(* Logix 5000 project; controller Amvex_Thorpe_Flowmeter vendor 1 type 14 code 106 rev 33.13; software revision 33.01; part 10 of 16 *)
(* tags used below, declared in another part *)
   FIRST_SCAN : BOOL;
   FIRST_SCAN_ONS : BOOL;
   ID86_InputDataLength : MESSAGE;   // Message Command Input Data Data Length
   ID86_LengthParameterdata : MESSAGE;   // Message Command Parameter Data Length
   ID86_MSG_Diagnostic : MESSAGE;   // Message Get Diagnosis Module
   ID86_MSG_ProcessAlarm : MESSAGE;   // Message Get Get Process Alram Module
   ID86_OutputDataLength : MESSAGE;   // Message Command Output Data Data Length
   ID86_ReceiveMSG1 : MESSAGE;   // Message Command Parameter Receive Data
   ID86_ReceiveMSG2 : MESSAGE;   // Message Command Parameter Receive Data
   ID86_ReceiveMSG3 : MESSAGE;   // Message Command Parameter Receive Data
   ID86_SendMSG1 : MESSAGE;   // Message Command Parameter Send Data
   ID86_SendMSG2 : MESSAGE;   // Message Command Parameter Send Data
   ID86_SendMSG3 : MESSAGE;   // Message Command Parameter Send Data
   MCP_00 : UDT_ID86;

PROGRAM MainProgram   (* main routine MainRoutine *)
VAR
   test : INT := 8;
END_VAR

ROUTINE MainRoutine   (* ladder *)
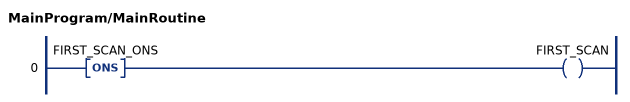
   0: ONS(FIRST_SCAN_ONS)OTE(FIRST_SCAN);
END_ROUTINE
END_PROGRAM

PROGRAM MCP_Main   (* main routine MAIN *)
VAR
   ActivateBtn : BOOL;
   Alicat0_ONS : BOOL;
   Alicat0DataInc : INT := 2;
   Alicat1_ONS : BOOL;
   Alicat1_ONS2 : BOOL := 1;
   Alicat1DataInc : INT := 7;
   Auto_Seq : SEQ := (Time_Out.PRE := 180000, Time_Out.ACC := 114179, Time_Out.EN := 1, Time_Out.TT := 1, Time_Out_Sec := 180);
   Barcode_Latch : BOOL;
   Barcode_ONS : BOOL;
   Barcode_Result_DATA : SINT[128] := ([0] := 69, [1] := 82, [2] := 82, [3] := 79, [4] := 82, [5] := 13, [6] := 56, [7] := 49, [8] := 48, [9] := 49, [10] := 53, [11] := 48, [12] := 51, [13] := 48, [14] := 48, [15] := 48, [16] := 50, [17] := 49, [18] := 84, [19] := 49, [20] := 53, [21] := 85, [22] := 79, [23] := 66, [24] := 51, [25] := 53, [26] := 48, [27] := 57, [28] := 56, [29] := 13);
   BarcodeSave_ons : BOOL;
   Counter_ONS : BOOL;
   debugtimer1 : TIMER := (PRE := 1000);
   DonePallets : COUNTER := (ACC := -70770);
   Fasttest_timer : TIMER := (PRE := 750);
   Fasttest_timer2 : TIMER := (PRE := 1000);
   FAULT : DINT;
   FAULTED : DINT;
   First_SEQ : BOOL;
   First_SEQ_ONS : BOOL;
   Flash_Timer_Off : TIMER := (PRE := 500);
   Flash_Timer_On : TIMER := (PRE := 500, ACC := 430, EN := 1, TT := 1);
   Gripper_ONS : BOOL;
   HMI_Counter_ONS : BOOL;
   Home_ONS : BOOL;
   HomeStep : INT;
   Infeed_Latch : BOOL;
   Infeed_ONS : BOOL := 1;
   InfeedPalletTM1 : TIMER := (PRE := 250);
   InfeedPalletTM2 : TIMER := (PRE := 250);
   IV3_Prog_AOI : IvSwichPrgoram := (TargetProgramNo := 3, SwitchProgramDone := 1);
   joggingONS : BOOL;
   Lift_stop_timer : TIMER := (PRE := 750);
   lift_stop_timer2 : TIMER := (PRE := 750);
   Manual_ONS : BOOL;
   Manual_Output_Reset : BOOL;
   MODE : MODE := (Manual := 1, Manual_ONS := 1, Selector := 2);
   Oxygen_TM : TIMER := (PRE := 500);
   PalletStop_ONS : BOOL;
   Part_count : DINT := 39;
   Prog_Switch_ons : BOOL;
   RCD_ONS : BOOL;
   RESET : BOOL;
   Rest_timer : TIMER := (PRE := 1000);
   RobotAngVel : SetCartAngVel := (Parameter_Value := 50.0);
   RobotConnected_ONS : BOOL;
   RobotConnection : BOOL;
   Setspeed : BOOL;
   SetupONS : BOOL;
   SR_Read_Complete_Clear : BOOL;
   SR_Read_Request : BOOL;
   SR_ReadSuccess : BOOL;
   Stopping_Latch : BOOL := 1;
   temp_Gripper_Delay : TIMER := (PRE := 250);
   Test : Connect;
   Test_Connection : Connect;
   Test_ONS : BOOL[32];
   Test_start_offline : StartOfflineProgram := (Parameter_Value := 1.0);
   test_Turn_ONS : BOOL;
   testing_ons : BOOL;
   testsstse : BOOL;
END_VAR

ROUTINE MAIN   (* ladder *)
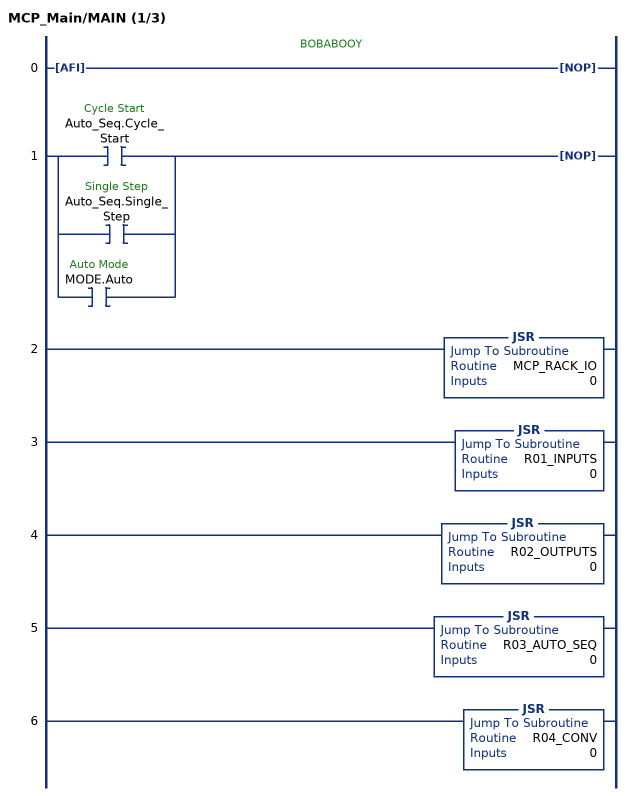
   // BOBABOOY
   0: AFI()NOP();
   1: [XIC(Auto_Seq.Cycle_Start) ,XIC(Auto_Seq.Single_Step) ,XIC(MODE.Auto) ]NOP();
   2: JSR(MCP_RACK_IO,0);
   3: JSR(R01_INPUTS,0);
   4: JSR(R02_OUTPUTS,0);
   5: JSR(R03_AUTO_SEQ,0);
   6: JSR(R04_CONV,0);
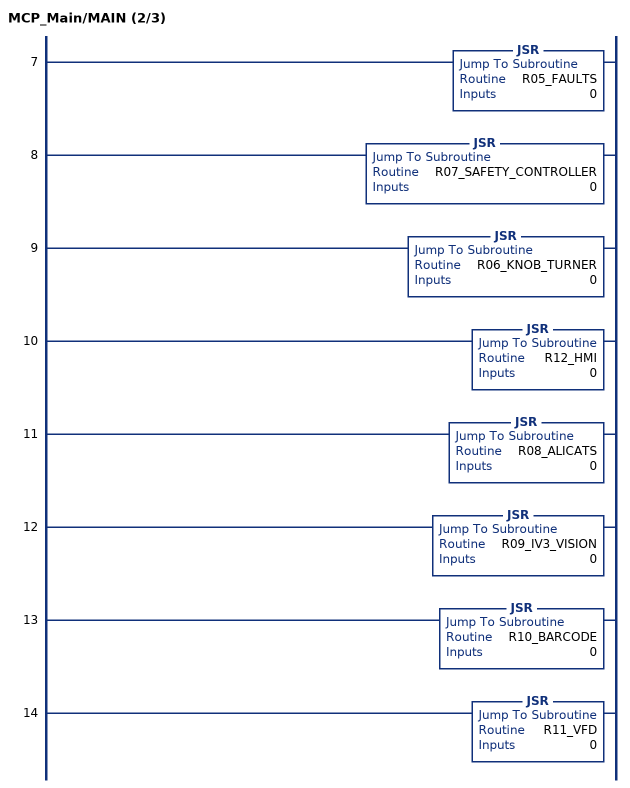
   7: JSR(R05_FAULTS,0);
   8: JSR(R07_SAFETY_CONTROLLER,0);
   9: JSR(R06_KNOB_TURNER,0);
   10: JSR(R12_HMI,0);
   11: JSR(R08_ALICATS,0);
   12: JSR(R09_IV3_VISION,0);
   13: JSR(R10_BARCODE,0);
   14: JSR(R11_VFD,0);
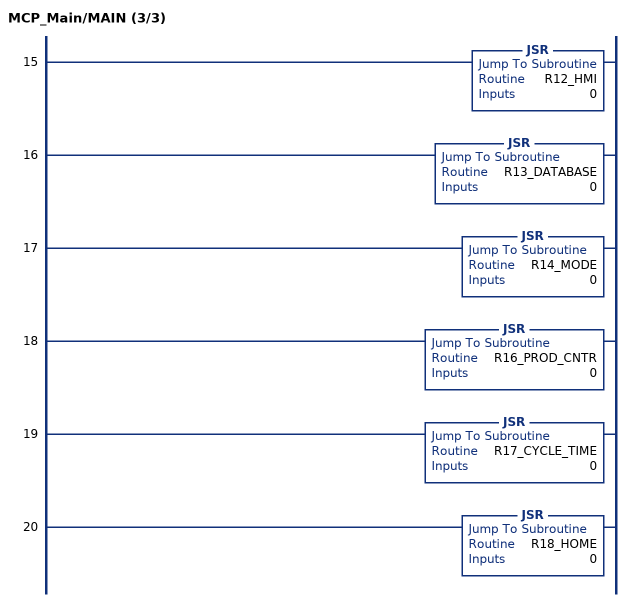
   15: JSR(R12_HMI,0);
   16: JSR(R13_DATABASE,0);
   17: JSR(R14_MODE,0);
   18: JSR(R16_PROD_CNTR,0);
   19: JSR(R17_CYCLE_TIME,0);
   20: JSR(R18_HOME,0);
END_ROUTINE

ROUTINE MCP_RACK_IO   (* ladder *)
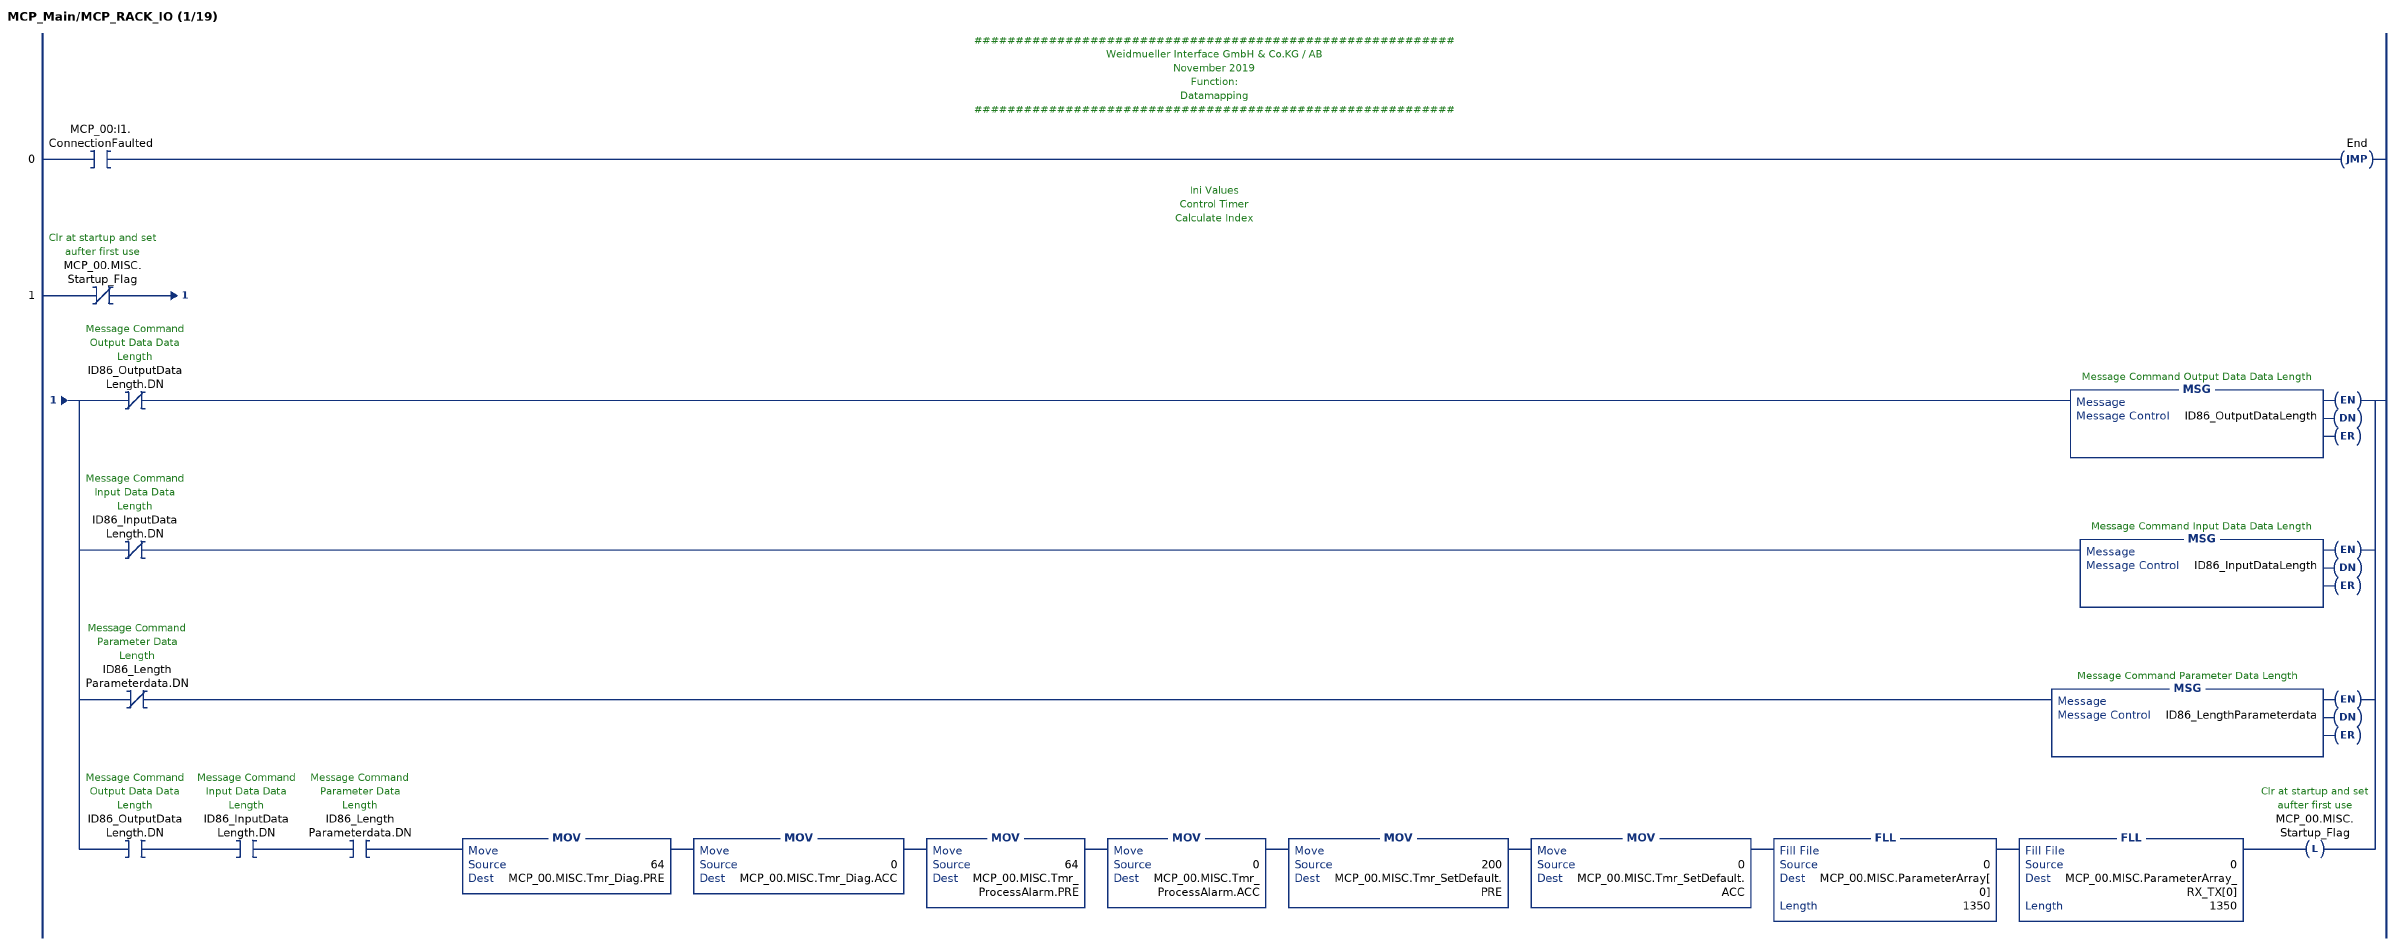
   // ##########################################################
   // Weidmueller Interface GmbH & Co.KG / AB
   // November 2019
   // Function:
   // Datamapping
   // ##########################################################
   0: XIC(MCP_00:I1.ConnectionFaulted)JMP(End);
   // Ini Values
   // Control Timer
   // Calculate Index
   1: XIO(MCP_00.MISC.Startup_Flag)[[XIO(ID86_OutputDataLength.DN) MSG(ID86_OutputDataLength) ,XIO(ID86_InputDataLength.DN) MSG(ID86_InputDataLength) ,XIO(ID86_LengthParameterdata.DN) MSG(ID86_LengthParameterdata) ] ,XIC(ID86_OutputDataLength.DN) XIC(ID86_InputDataLength.DN) XIC(ID86_LengthParameterdata.DN) MOV(64,MCP_00.MISC.Tmr_Diag.PRE) MOV(0,MCP_00.MISC.Tmr_Diag.ACC) MOV(64,MCP_00.MISC.Tmr_ProcessAlarm.PRE) MOV(0,MCP_00.MISC.Tmr_ProcessAlarm.ACC) MOV(200,MCP_00.MISC.Tmr_SetDefault.PRE) MOV(0,MCP_00.MISC.Tmr_SetDefault.ACC) FLL(0,MCP_00.MISC.ParameterArray[0],1350) FLL(0,MCP_00.MISC.ParameterArray_RX_TX[0],1350) OTL(MCP_00.MISC.Startup_Flag) ];
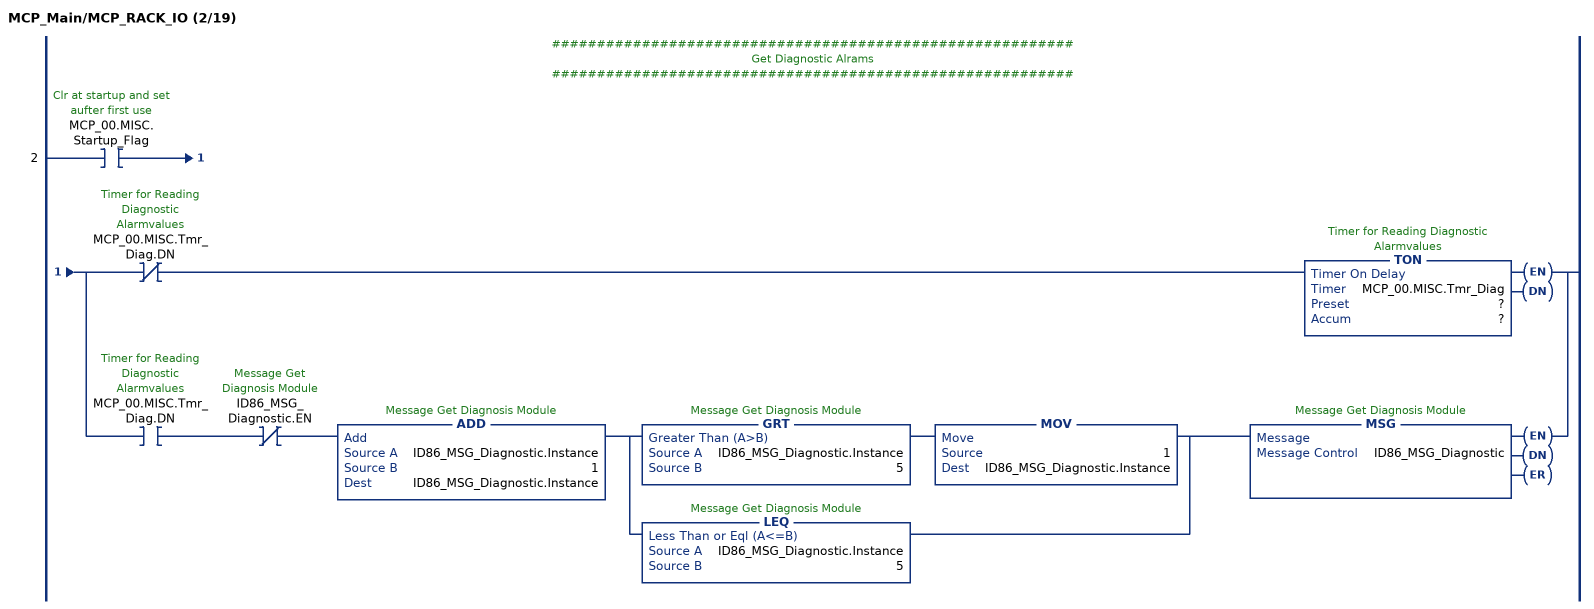
   // ##########################################################
   // Get Diagnostic Alrams
   // ##########################################################
   2: XIC(MCP_00.MISC.Startup_Flag)[XIO(MCP_00.MISC.Tmr_Diag.DN) TON(MCP_00.MISC.Tmr_Diag,?,?) ,XIC(MCP_00.MISC.Tmr_Diag.DN) XIO(ID86_MSG_Diagnostic.EN) ADD(ID86_MSG_Diagnostic.Instance,1,ID86_MSG_Diagnostic.Instance) [GRT(ID86_MSG_Diagnostic.Instance,5) MOV(1,ID86_MSG_Diagnostic.Instance) ,LEQ(ID86_MSG_Diagnostic.Instance,5) ] MSG(ID86_MSG_Diagnostic) ];
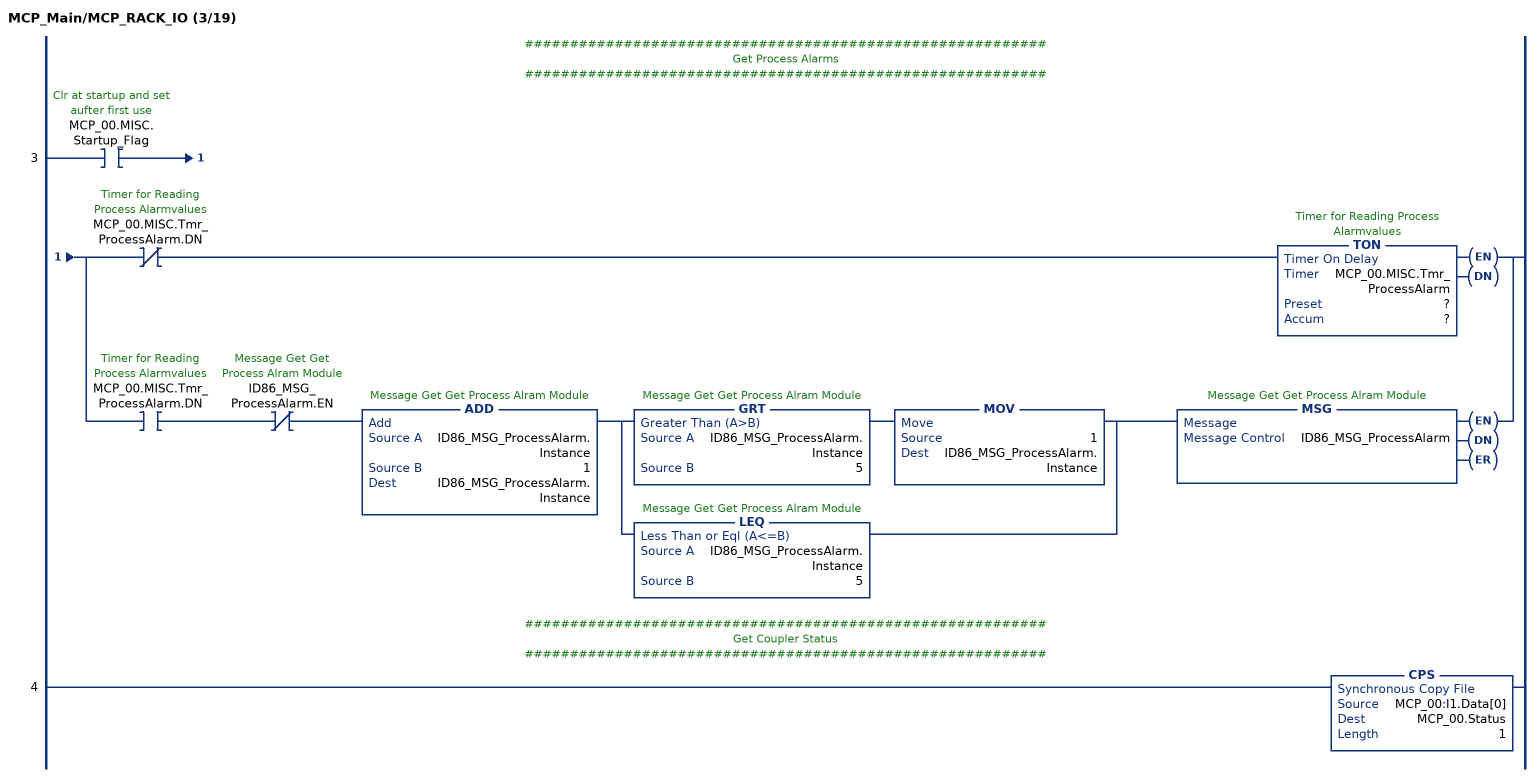
   // ##########################################################
   // Get Process Alarms
   // ##########################################################
   3: XIC(MCP_00.MISC.Startup_Flag)[XIO(MCP_00.MISC.Tmr_ProcessAlarm.DN) TON(MCP_00.MISC.Tmr_ProcessAlarm,?,?) ,XIC(MCP_00.MISC.Tmr_ProcessAlarm.DN) XIO(ID86_MSG_ProcessAlarm.EN) ADD(ID86_MSG_ProcessAlarm.Instance,1,ID86_MSG_ProcessAlarm.Instance) [GRT(ID86_MSG_ProcessAlarm.Instance,5) MOV(1,ID86_MSG_ProcessAlarm.Instance) ,LEQ(ID86_MSG_ProcessAlarm.Instance,5) ] MSG(ID86_MSG_ProcessAlarm) ];
   // ##########################################################
   // Get Coupler Status
   // ##########################################################
   4: CPS(MCP_00:I1.Data[0],MCP_00.Status,1);
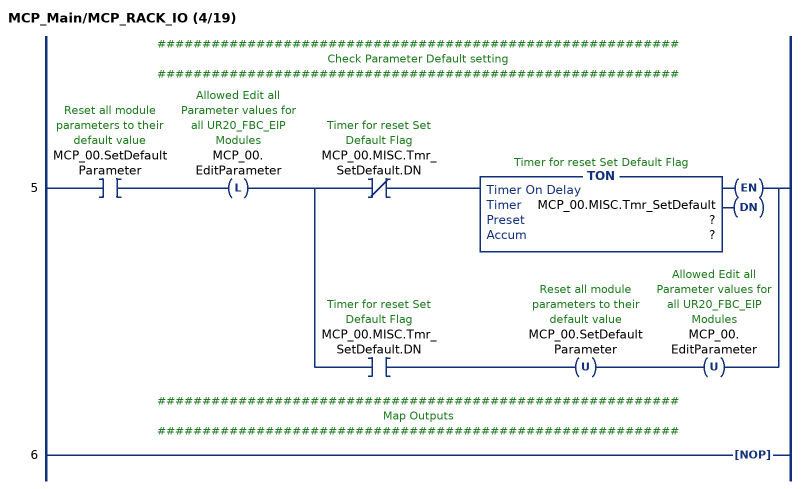
   // ##########################################################
   // Check Parameter Default setting
   // ##########################################################
   5: XIC(MCP_00.SetDefaultParameter)OTL(MCP_00.EditParameter)[XIO(MCP_00.MISC.Tmr_SetDefault.DN) TON(MCP_00.MISC.Tmr_SetDefault,?,?) ,XIC(MCP_00.MISC.Tmr_SetDefault.DN) OTU(MCP_00.SetDefaultParameter) OTU(MCP_00.EditParameter) ];
   // ##########################################################
   // Map Outputs
   // ##########################################################
   6: NOP();
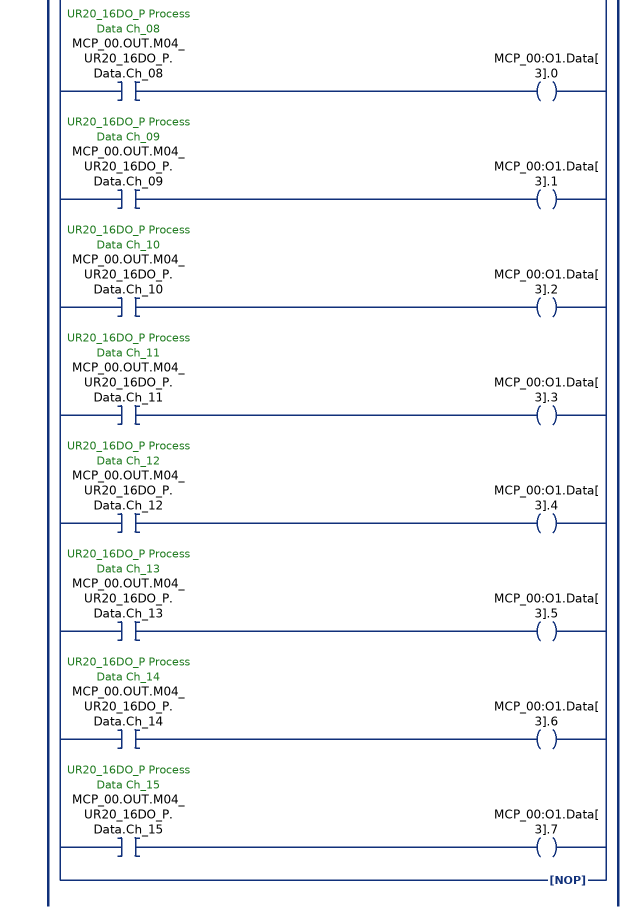
   // Map
   //  UR20_16DO_P
   //  Module No 4
   //  Process Data
   //  Outputs
   7: [NOP() ,XIC(MCP_00.OUT.M04_UR20_16DO_P.Data.Ch_00) OTE(MCP_00:O1.Data[2].0) ,XIC(MCP_00.OUT.M04_UR20_16DO_P.Data.Ch_01) OTE(MCP_00:O1.Data[2].1) ,XIC(MCP_00.OUT.M04_UR20_16DO_P.Data.Ch_02) OTE(MCP_00:O1.Data[2].2) ,XIC(MCP_00.OUT.M04_UR20_16DO_P.Data.Ch_03) OTE(MCP_00:O1.Data[2].3) ,XIC(MCP_00.OUT.M04_UR20_16DO_P.Data.Ch_04) OTE(MCP_00:O1.Data[2].4) ,XIC(MCP_00.OUT.M04_UR20_16DO_P.Data.Ch_05) OTE(MCP_00:O1.Data[2].5) ,XIC(MCP_00.OUT.M04_UR20_16DO_P.Data.Ch_06) OTE(MCP_00:O1.Data[2].6) ,XIC(MCP_00.OUT.M04_UR20_16DO_P.Data.Ch_07) OTE(MCP_00:O1.Data[2].7) ,XIC(MCP_00.OUT.M04_UR20_16DO_P.Data.Ch_08) OTE(MCP_00:O1.Data[3].0) ,XIC(MCP_00.OUT.M04_UR20_16DO_P.Data.Ch_09) OTE(MCP_00:O1.Data[3].1) ,XIC(MCP_00.OUT.M04_UR20_16DO_P.Data.Ch_10) OTE(MCP_00:O1.Data[3].2) ,XIC(MCP_00.OUT.M04_UR20_16DO_P.Data.Ch_11) OTE(MCP_00:O1.Data[3].3) ,XIC(MCP_00.OUT.M04_UR20_16DO_P.Data.Ch_12) OTE(MCP_00:O1.Data[3].4) ,XIC(MCP_00.OUT.M04_UR20_16DO_P.Data.Ch_13) OTE(MCP_00:O1.Data[3].5) ,XIC(MCP_00.OUT.M04_UR20_16DO_P.Data.Ch_14) OTE(MCP_00:O1.Data[3].6) ,XIC(MCP_00.OUT.M04_UR20_16DO_P.Data.Ch_15) OTE(MCP_00:O1.Data[3].7) ,NOP() ];
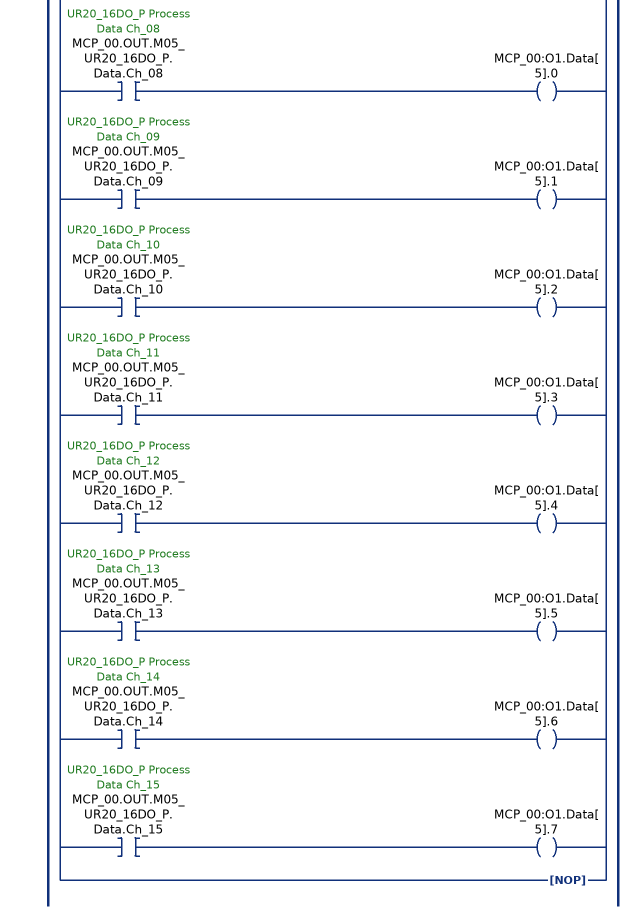
   // Map
   //  UR20_16DO_P
   //  Module No 5
   //  Process Data
   //  Outputs
   8: [NOP() ,XIC(MCP_00.OUT.M05_UR20_16DO_P.Data.Ch_00) OTE(MCP_00:O1.Data[4].0) ,XIC(MCP_00.OUT.M05_UR20_16DO_P.Data.Ch_01) OTE(MCP_00:O1.Data[4].1) ,XIC(MCP_00.OUT.M05_UR20_16DO_P.Data.Ch_02) OTE(MCP_00:O1.Data[4].2) ,XIC(MCP_00.OUT.M05_UR20_16DO_P.Data.Ch_03) OTE(MCP_00:O1.Data[4].3) ,XIC(MCP_00.OUT.M05_UR20_16DO_P.Data.Ch_04) OTE(MCP_00:O1.Data[4].4) ,XIC(MCP_00.OUT.M05_UR20_16DO_P.Data.Ch_05) OTE(MCP_00:O1.Data[4].5) ,XIC(MCP_00.OUT.M05_UR20_16DO_P.Data.Ch_06) OTE(MCP_00:O1.Data[4].6) ,XIC(MCP_00.OUT.M05_UR20_16DO_P.Data.Ch_07) OTE(MCP_00:O1.Data[4].7) ,XIC(MCP_00.OUT.M05_UR20_16DO_P.Data.Ch_08) OTE(MCP_00:O1.Data[5].0) ,XIC(MCP_00.OUT.M05_UR20_16DO_P.Data.Ch_09) OTE(MCP_00:O1.Data[5].1) ,XIC(MCP_00.OUT.M05_UR20_16DO_P.Data.Ch_10) OTE(MCP_00:O1.Data[5].2) ,XIC(MCP_00.OUT.M05_UR20_16DO_P.Data.Ch_11) OTE(MCP_00:O1.Data[5].3) ,XIC(MCP_00.OUT.M05_UR20_16DO_P.Data.Ch_12) OTE(MCP_00:O1.Data[5].4) ,XIC(MCP_00.OUT.M05_UR20_16DO_P.Data.Ch_13) OTE(MCP_00:O1.Data[5].5) ,XIC(MCP_00.OUT.M05_UR20_16DO_P.Data.Ch_14) OTE(MCP_00:O1.Data[5].6) ,XIC(MCP_00.OUT.M05_UR20_16DO_P.Data.Ch_15) OTE(MCP_00:O1.Data[5].7) ,NOP() ];
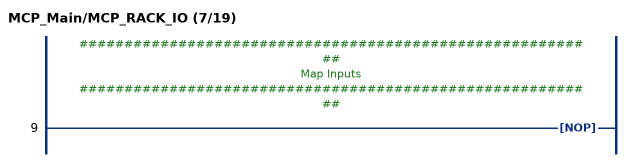
   // ##########################################################
   // Map Inputs
   // ##########################################################
   9: NOP();
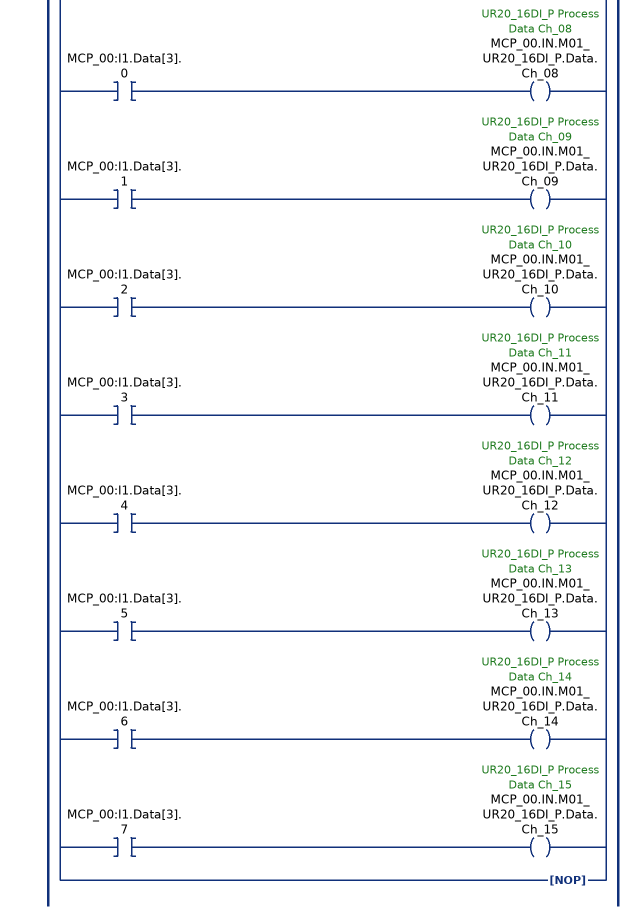
   // Map
   //  UR20_16DI_P
   //  Module No 1
   //  Process Data
   //  Inputs
   10: [NOP() ,XIC(MCP_00:I1.Data[2].0) OTE(MCP_00.IN.M01_UR20_16DI_P.Data.Ch_00) ,XIC(MCP_00:I1.Data[2].1) OTE(MCP_00.IN.M01_UR20_16DI_P.Data.Ch_01) ,XIC(MCP_00:I1.Data[2].2) OTE(MCP_00.IN.M01_UR20_16DI_P.Data.Ch_02) ,XIC(MCP_00:I1.Data[2].3) OTE(MCP_00.IN.M01_UR20_16DI_P.Data.Ch_03) ,XIC(MCP_00:I1.Data[2].4) OTE(MCP_00.IN.M01_UR20_16DI_P.Data.Ch_04) ,XIC(MCP_00:I1.Data[2].5) OTE(MCP_00.IN.M01_UR20_16DI_P.Data.Ch_05) ,XIC(MCP_00:I1.Data[2].6) OTE(MCP_00.IN.M01_UR20_16DI_P.Data.Ch_06) ,XIC(MCP_00:I1.Data[2].7) OTE(MCP_00.IN.M01_UR20_16DI_P.Data.Ch_07) ,XIC(MCP_00:I1.Data[3].0) OTE(MCP_00.IN.M01_UR20_16DI_P.Data.Ch_08) ,XIC(MCP_00:I1.Data[3].1) OTE(MCP_00.IN.M01_UR20_16DI_P.Data.Ch_09) ,XIC(MCP_00:I1.Data[3].2) OTE(MCP_00.IN.M01_UR20_16DI_P.Data.Ch_10) ,XIC(MCP_00:I1.Data[3].3) OTE(MCP_00.IN.M01_UR20_16DI_P.Data.Ch_11) ,XIC(MCP_00:I1.Data[3].4) OTE(MCP_00.IN.M01_UR20_16DI_P.Data.Ch_12) ,XIC(MCP_00:I1.Data[3].5) OTE(MCP_00.IN.M01_UR20_16DI_P.Data.Ch_13) ,XIC(MCP_00:I1.Data[3].6) OTE(MCP_00.IN.M01_UR20_16DI_P.Data.Ch_14) ,XIC(MCP_00:I1.Data[3].7) OTE(MCP_00.IN.M01_UR20_16DI_P.Data.Ch_15) ,NOP() ];
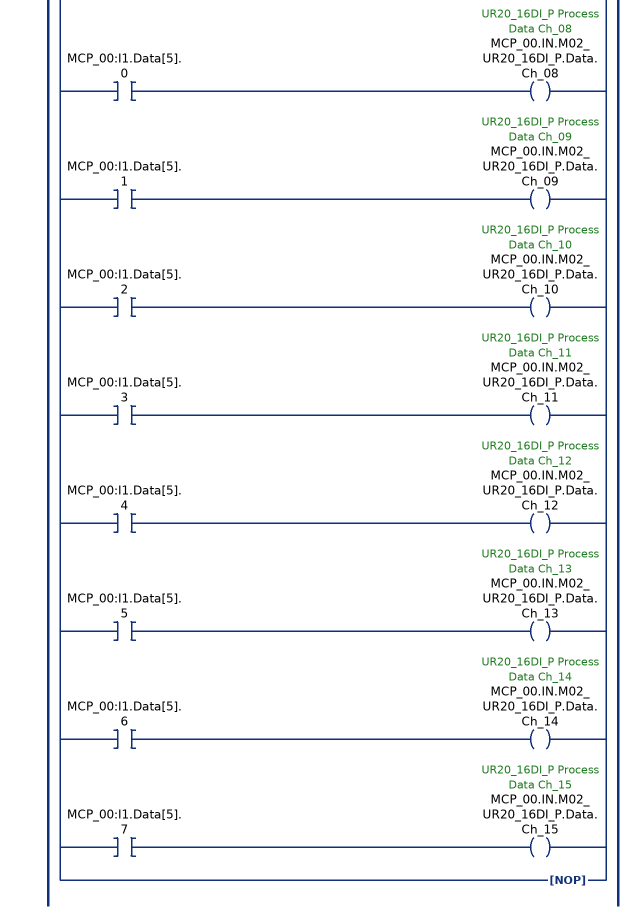
   // Map
   //  UR20_16DI_P
   //  Module No 2
   //  Process Data
   //  Inputs
   11: [NOP() ,XIC(MCP_00:I1.Data[4].0) OTE(MCP_00.IN.M02_UR20_16DI_P.Data.Ch_00) ,XIC(MCP_00:I1.Data[4].1) OTE(MCP_00.IN.M02_UR20_16DI_P.Data.Ch_01) ,XIC(MCP_00:I1.Data[4].2) OTE(MCP_00.IN.M02_UR20_16DI_P.Data.Ch_02) ,XIC(MCP_00:I1.Data[4].3) OTE(MCP_00.IN.M02_UR20_16DI_P.Data.Ch_03) ,XIC(MCP_00:I1.Data[4].4) OTE(MCP_00.IN.M02_UR20_16DI_P.Data.Ch_04) ,XIC(MCP_00:I1.Data[4].5) OTE(MCP_00.IN.M02_UR20_16DI_P.Data.Ch_05) ,XIC(MCP_00:I1.Data[4].6) OTE(MCP_00.IN.M02_UR20_16DI_P.Data.Ch_06) ,XIC(MCP_00:I1.Data[4].7) OTE(MCP_00.IN.M02_UR20_16DI_P.Data.Ch_07) ,XIC(MCP_00:I1.Data[5].0) OTE(MCP_00.IN.M02_UR20_16DI_P.Data.Ch_08) ,XIC(MCP_00:I1.Data[5].1) OTE(MCP_00.IN.M02_UR20_16DI_P.Data.Ch_09) ,XIC(MCP_00:I1.Data[5].2) OTE(MCP_00.IN.M02_UR20_16DI_P.Data.Ch_10) ,XIC(MCP_00:I1.Data[5].3) OTE(MCP_00.IN.M02_UR20_16DI_P.Data.Ch_11) ,XIC(MCP_00:I1.Data[5].4) OTE(MCP_00.IN.M02_UR20_16DI_P.Data.Ch_12) ,XIC(MCP_00:I1.Data[5].5) OTE(MCP_00.IN.M02_UR20_16DI_P.Data.Ch_13) ,XIC(MCP_00:I1.Data[5].6) OTE(MCP_00.IN.M02_UR20_16DI_P.Data.Ch_14) ,XIC(MCP_00:I1.Data[5].7) OTE(MCP_00.IN.M02_UR20_16DI_P.Data.Ch_15) ,NOP() ];
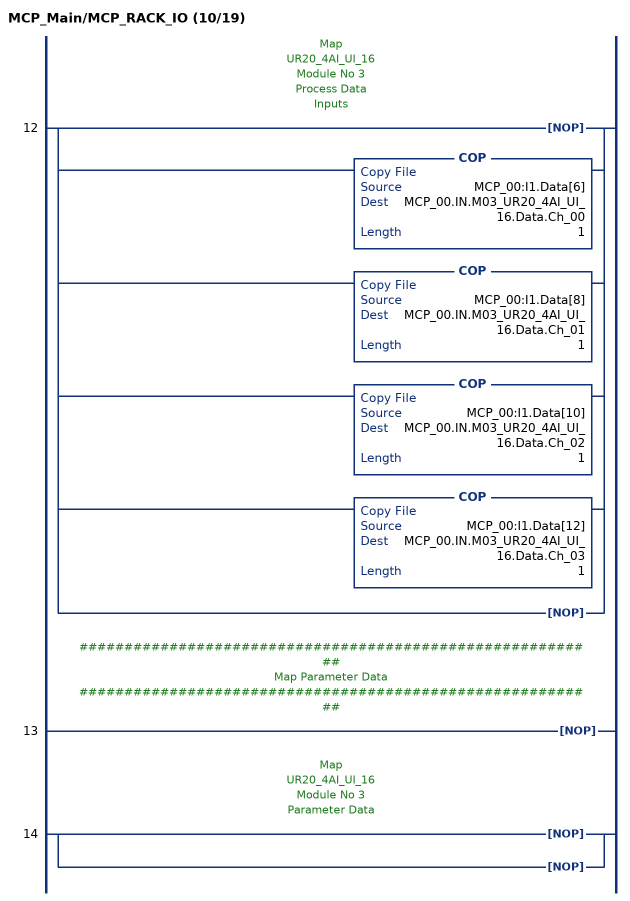
   // Map
   //  UR20_4AI_UI_16
   //  Module No 3
   //  Process Data
   //  Inputs
   12: [NOP() ,COP(MCP_00:I1.Data[6],MCP_00.IN.M03_UR20_4AI_UI_16.Data.Ch_00,1) ,COP(MCP_00:I1.Data[8],MCP_00.IN.M03_UR20_4AI_UI_16.Data.Ch_01,1) ,COP(MCP_00:I1.Data[10],MCP_00.IN.M03_UR20_4AI_UI_16.Data.Ch_02,1) ,COP(MCP_00:I1.Data[12],MCP_00.IN.M03_UR20_4AI_UI_16.Data.Ch_03,1) ,NOP() ];
   // ##########################################################
   // Map Parameter Data
   // ##########################################################
   13: NOP();
   // Map
   //  UR20_4AI_UI_16
   //  Module No 3
   //  Parameter Data
   14: [NOP() ,NOP() ];
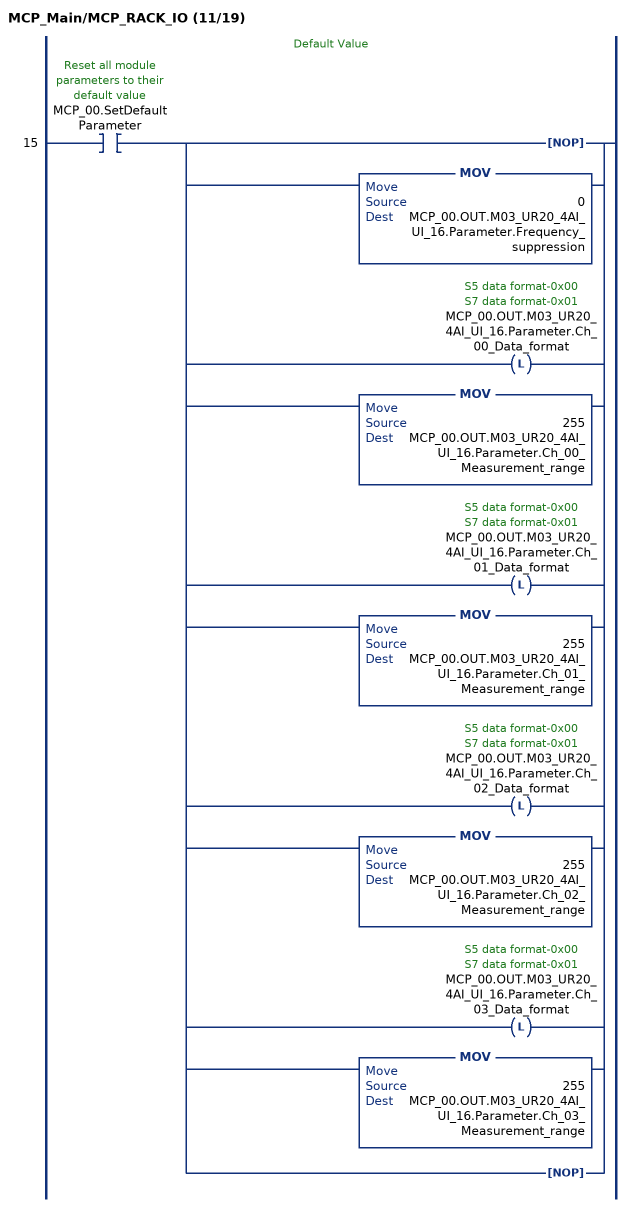
   // Default Value
   15: XIC(MCP_00.SetDefaultParameter)[NOP() ,MOV(0,MCP_00.OUT.M03_UR20_4AI_UI_16.Parameter.Frequency_suppression) ,OTL(MCP_00.OUT.M03_UR20_4AI_UI_16.Parameter.Ch_00_Data_format) ,MOV(255,MCP_00.OUT.M03_UR20_4AI_UI_16.Parameter.Ch_00_Measurement_range) ,OTL(MCP_00.OUT.M03_UR20_4AI_UI_16.Parameter.Ch_01_Data_format) ,MOV(255,MCP_00.OUT.M03_UR20_4AI_UI_16.Parameter.Ch_01_Measurement_range) ,OTL(MCP_00.OUT.M03_UR20_4AI_UI_16.Parameter.Ch_02_Data_format) ,MOV(255,MCP_00.OUT.M03_UR20_4AI_UI_16.Parameter.Ch_02_Measurement_range) ,OTL(MCP_00.OUT.M03_UR20_4AI_UI_16.Parameter.Ch_03_Data_format) ,MOV(255,MCP_00.OUT.M03_UR20_4AI_UI_16.Parameter.Ch_03_Measurement_range) ,NOP() ];
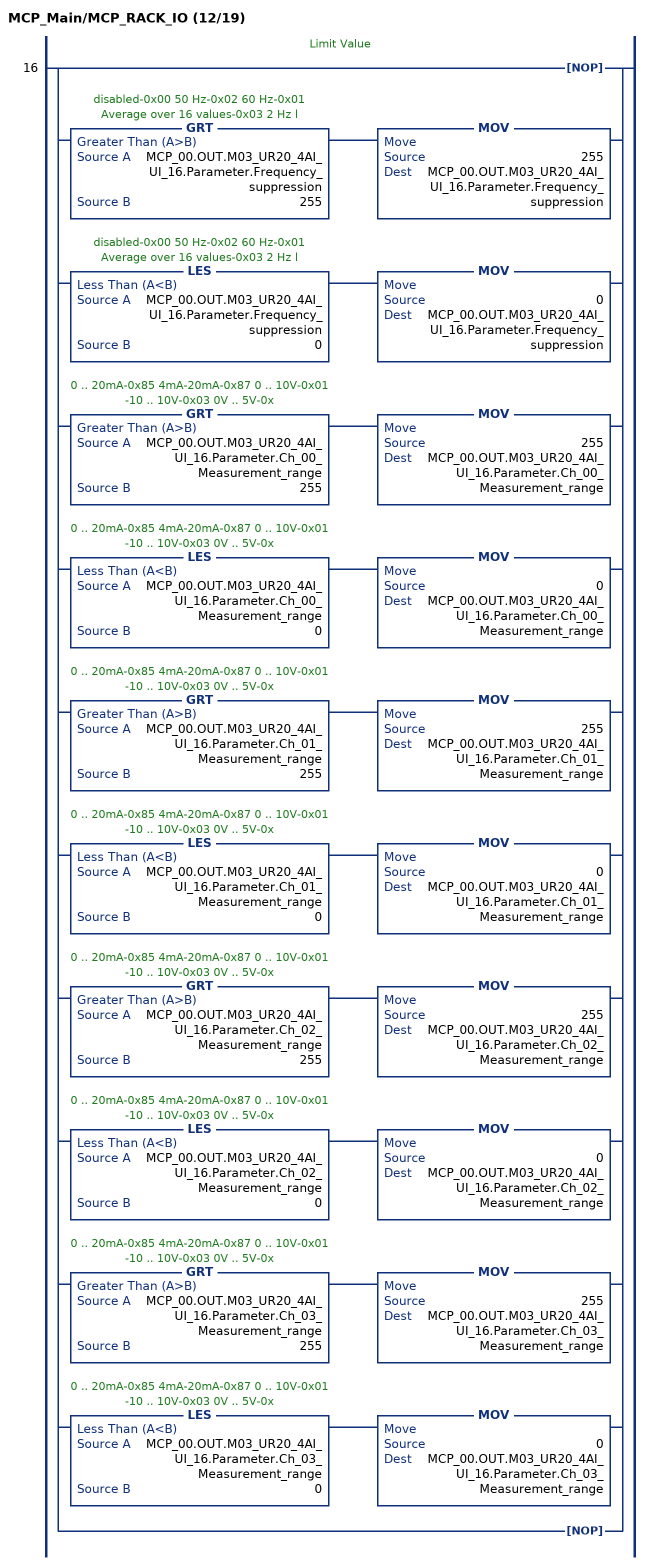
   // Limit Value
   16: [NOP() ,GRT(MCP_00.OUT.M03_UR20_4AI_UI_16.Parameter.Frequency_suppression,255) MOV(255,MCP_00.OUT.M03_UR20_4AI_UI_16.Parameter.Frequency_suppression) ,LES(MCP_00.OUT.M03_UR20_4AI_UI_16.Parameter.Frequency_suppression,0) MOV(0,MCP_00.OUT.M03_UR20_4AI_UI_16.Parameter.Frequency_suppression) ,GRT(MCP_00.OUT.M03_UR20_4AI_UI_16.Parameter.Ch_00_Measurement_range,255) MOV(255,MCP_00.OUT.M03_UR20_4AI_UI_16.Parameter.Ch_00_Measurement_range) ,LES(MCP_00.OUT.M03_UR20_4AI_UI_16.Parameter.Ch_00_Measurement_range,0) MOV(0,MCP_00.OUT.M03_UR20_4AI_UI_16.Parameter.Ch_00_Measurement_range) ,GRT(MCP_00.OUT.M03_UR20_4AI_UI_16.Parameter.Ch_01_Measurement_range,255) MOV(255,MCP_00.OUT.M03_UR20_4AI_UI_16.Parameter.Ch_01_Measurement_range) ,LES(MCP_00.OUT.M03_UR20_4AI_UI_16.Parameter.Ch_01_Measurement_range,0) MOV(0,MCP_00.OUT.M03_UR20_4AI_UI_16.Parameter.Ch_01_Measurement_range) ,GRT(MCP_00.OUT.M03_UR20_4AI_UI_16.Parameter.Ch_02_Measurement_range,255) MOV(255,MCP_00.OUT.M03_UR20_4AI_UI_16.Parameter.Ch_02_Measurement_range) ,LES(MCP_00.OUT.M03_UR20_4AI_UI_16.Parameter.Ch_02_Measurement_range,0) MOV(0,MCP_00.OUT.M03_UR20_4AI_UI_16.Parameter.Ch_02_Measurement_range) ,GRT(MCP_00.OUT.M03_UR20_4AI_UI_16.Parameter.Ch_03_Measurement_range,255) MOV(255,MCP_00.OUT.M03_UR20_4AI_UI_16.Parameter.Ch_03_Measurement_range) ,LES(MCP_00.OUT.M03_UR20_4AI_UI_16.Parameter.Ch_03_Measurement_range,0) MOV(0,MCP_00.OUT.M03_UR20_4AI_UI_16.Parameter.Ch_03_Measurement_range) ,NOP() ];
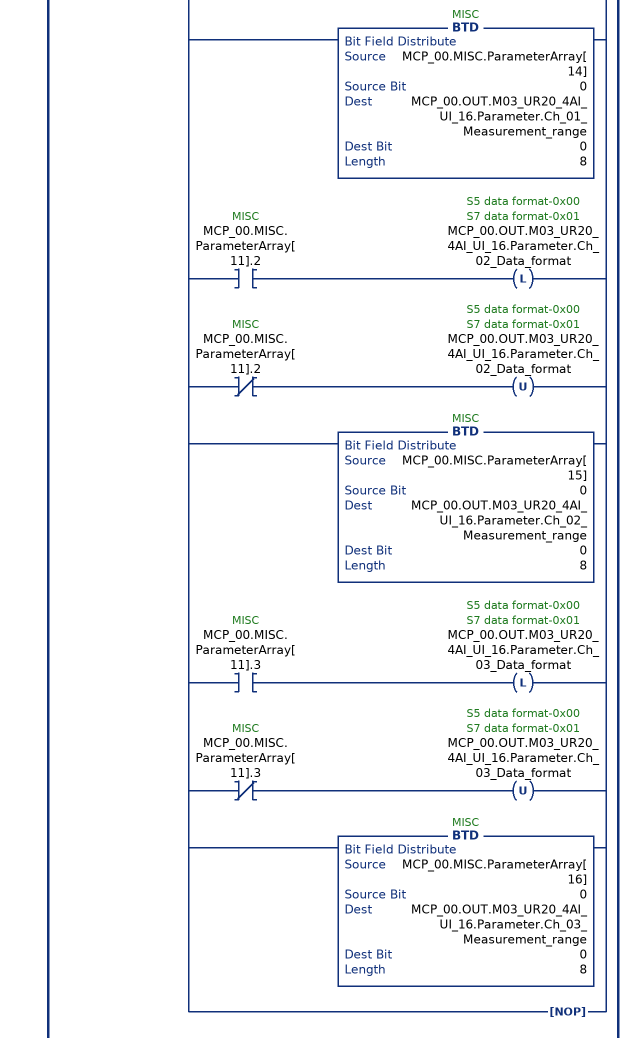
   // Read Parameter from Module
   17: XIO(MCP_00.EditParameter)[NOP() ,BTD(MCP_00.MISC.ParameterArray[12],0,MCP_00.OUT.M03_UR20_4AI_UI_16.Parameter.Frequency_suppression,0,8) ,XIC(MCP_00.MISC.ParameterArray[11].0) OTL(MCP_00.OUT.M03_UR20_4AI_UI_16.Parameter.Ch_00_Data_format) ,XIO(MCP_00.MISC.ParameterArray[11].0) OTU(MCP_00.OUT.M03_UR20_4AI_UI_16.Parameter.Ch_00_Data_format) ,BTD(MCP_00.MISC.ParameterArray[13],0,MCP_00.OUT.M03_UR20_4AI_UI_16.Parameter.Ch_00_Measurement_range,0,8) ,XIC(MCP_00.MISC.ParameterArray[11].1) OTL(MCP_00.OUT.M03_UR20_4AI_UI_16.Parameter.Ch_01_Data_format) ,XIO(MCP_00.MISC.ParameterArray[11].1) OTU(MCP_00.OUT.M03_UR20_4AI_UI_16.Parameter.Ch_01_Data_format) ,BTD(MCP_00.MISC.ParameterArray[14],0,MCP_00.OUT.M03_UR20_4AI_UI_16.Parameter.Ch_01_Measurement_range,0,8) ,XIC(MCP_00.MISC.ParameterArray[11].2) OTL(MCP_00.OUT.M03_UR20_4AI_UI_16.Parameter.Ch_02_Data_format) ,XIO(MCP_00.MISC.ParameterArray[11].2) OTU(MCP_00.OUT.M03_UR20_4AI_UI_16.Parameter.Ch_02_Data_format) ,BTD(MCP_00.MISC.ParameterArray[15],0,MCP_00.OUT.M03_UR20_4AI_UI_16.Parameter.Ch_02_Measurement_range,0,8) ,XIC(MCP_00.MISC.ParameterArray[11].3) OTL(MCP_00.OUT.M03_UR20_4AI_UI_16.Parameter.Ch_03_Data_format) ,XIO(MCP_00.MISC.ParameterArray[11].3) OTU(MCP_00.OUT.M03_UR20_4AI_UI_16.Parameter.Ch_03_Data_format) ,BTD(MCP_00.MISC.ParameterArray[16],0,MCP_00.OUT.M03_UR20_4AI_UI_16.Parameter.Ch_03_Measurement_range,0,8) ,NOP() ];
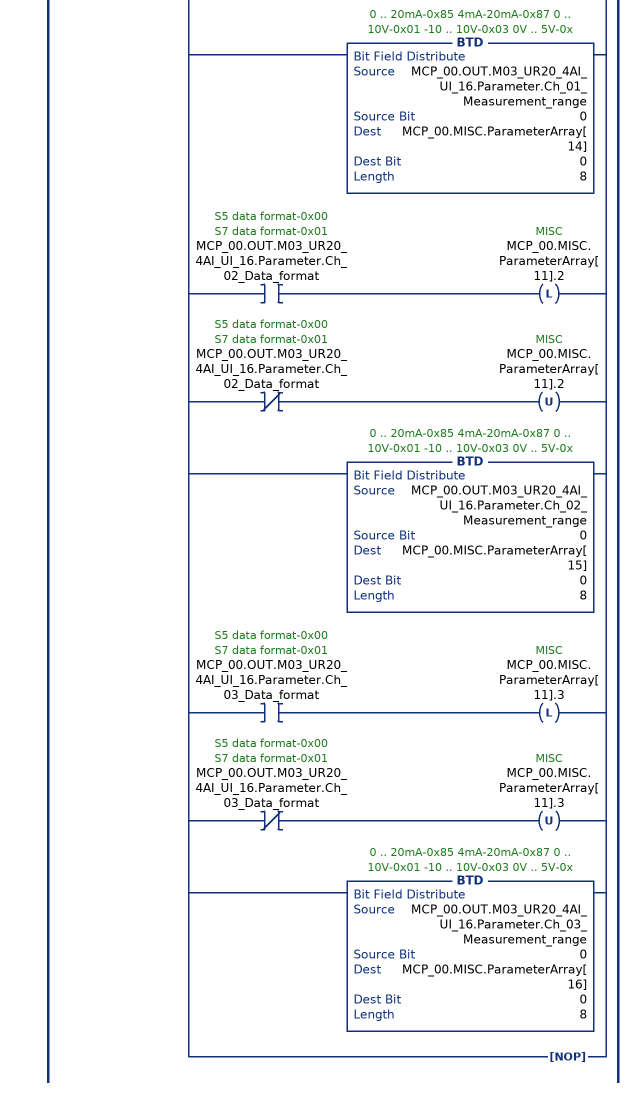
   // Write Parameter to Module
   18: XIC(MCP_00.EditParameter)[NOP() ,BTD(MCP_00.OUT.M03_UR20_4AI_UI_16.Parameter.Frequency_suppression,0,MCP_00.MISC.ParameterArray[12],0,8) ,XIC(MCP_00.OUT.M03_UR20_4AI_UI_16.Parameter.Ch_00_Data_format) OTL(MCP_00.MISC.ParameterArray[11].0) ,XIO(MCP_00.OUT.M03_UR20_4AI_UI_16.Parameter.Ch_00_Data_format) OTU(MCP_00.MISC.ParameterArray[11].0) ,BTD(MCP_00.OUT.M03_UR20_4AI_UI_16.Parameter.Ch_00_Measurement_range,0,MCP_00.MISC.ParameterArray[13],0,8) ,XIC(MCP_00.OUT.M03_UR20_4AI_UI_16.Parameter.Ch_01_Data_format) OTL(MCP_00.MISC.ParameterArray[11].1) ,XIO(MCP_00.OUT.M03_UR20_4AI_UI_16.Parameter.Ch_01_Data_format) OTU(MCP_00.MISC.ParameterArray[11].1) ,BTD(MCP_00.OUT.M03_UR20_4AI_UI_16.Parameter.Ch_01_Measurement_range,0,MCP_00.MISC.ParameterArray[14],0,8) ,XIC(MCP_00.OUT.M03_UR20_4AI_UI_16.Parameter.Ch_02_Data_format) OTL(MCP_00.MISC.ParameterArray[11].2) ,XIO(MCP_00.OUT.M03_UR20_4AI_UI_16.Parameter.Ch_02_Data_format) OTU(MCP_00.MISC.ParameterArray[11].2) ,BTD(MCP_00.OUT.M03_UR20_4AI_UI_16.Parameter.Ch_02_Measurement_range,0,MCP_00.MISC.ParameterArray[15],0,8) ,XIC(MCP_00.OUT.M03_UR20_4AI_UI_16.Parameter.Ch_03_Data_format) OTL(MCP_00.MISC.ParameterArray[11].3) ,XIO(MCP_00.OUT.M03_UR20_4AI_UI_16.Parameter.Ch_03_Data_format) OTU(MCP_00.MISC.ParameterArray[11].3) ,BTD(MCP_00.OUT.M03_UR20_4AI_UI_16.Parameter.Ch_03_Measurement_range,0,MCP_00.MISC.ParameterArray[16],0,8) ,NOP() ];
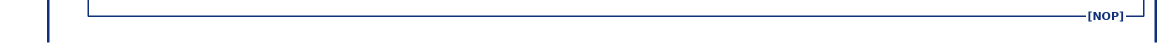
   // ##########################################################
   // DiagnoseAlarm Daten
   // ##########################################################
   19: XIC(ID86_MSG_Diagnostic.DN)[NOP() ,EQU(ID86_MSG_Diagnostic.Instance,1) [NEQ(MCP_00.MISC.DiagnosticData[0],0) OTL(MCP_00.IN.M01_UR20_16DI_P.StatusDiagAlarm) ,EQU(MCP_00.MISC.DiagnosticData[0],0) OTU(MCP_00.IN.M01_UR20_16DI_P.StatusDiagAlarm) ] CPS(MCP_00.MISC.DiagnosticData[0],MCP_00.IN.M01_UR20_16DI_P.Diagnostic,1) ,EQU(ID86_MSG_Diagnostic.Instance,2) [NEQ(MCP_00.MISC.DiagnosticData[0],0) OTL(MCP_00.IN.M02_UR20_16DI_P.StatusDiagAlarm) ,EQU(MCP_00.MISC.DiagnosticData[0],0) OTU(MCP_00.IN.M02_UR20_16DI_P.StatusDiagAlarm) ] CPS(MCP_00.MISC.DiagnosticData[0],MCP_00.IN.M02_UR20_16DI_P.Diagnostic,1) ,EQU(ID86_MSG_Diagnostic.Instance,3) [NEQ(MCP_00.MISC.DiagnosticData[0],0) OTL(MCP_00.IN.M03_UR20_4AI_UI_16.StatusDiagAlarm) ,EQU(MCP_00.MISC.DiagnosticData[0],0) OTU(MCP_00.IN.M03_UR20_4AI_UI_16.StatusDiagAlarm) ] CPS(MCP_00.MISC.DiagnosticData[0],MCP_00.IN.M03_UR20_4AI_UI_16.Diagnostic,1) ,EQU(ID86_MSG_Diagnostic.Instance,4) [NEQ(MCP_00.MISC.DiagnosticData[0],0) OTL(MCP_00.IN.M04_UR20_16DO_P.StatusDiagAlarm) ,EQU(MCP_00.MISC.DiagnosticData[0],0) OTU(MCP_00.IN.M04_UR20_16DO_P.StatusDiagAlarm) ] CPS(MCP_00.MISC.DiagnosticData[0],MCP_00.IN.M04_UR20_16DO_P.Diagnostic,1) ,EQU(ID86_MSG_Diagnostic.Instance,5) [NEQ(MCP_00.MISC.DiagnosticData[0],0) OTL(MCP_00.IN.M05_UR20_16DO_P.StatusDiagAlarm) ,EQU(MCP_00.MISC.DiagnosticData[0],0) OTU(MCP_00.IN.M05_UR20_16DO_P.StatusDiagAlarm) ] CPS(MCP_00.MISC.DiagnosticData[0],MCP_00.IN.M05_UR20_16DO_P.Diagnostic,1) ,NOP() ];
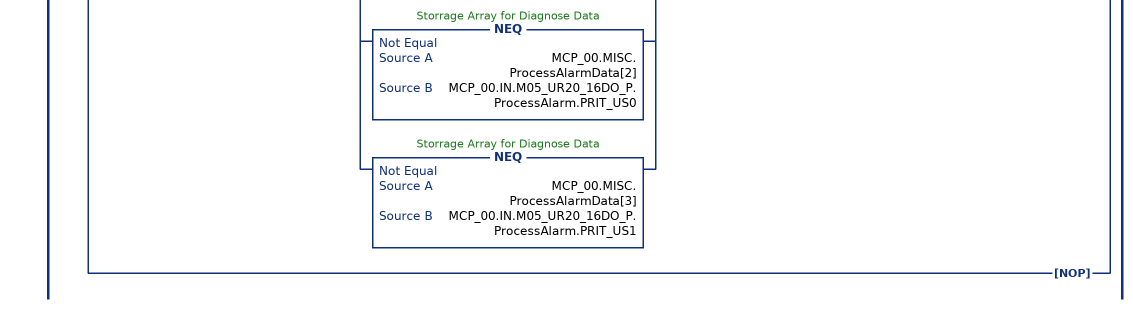
   // ##########################################################
   // ProcessAlarm Daten
   // ##########################################################
   20: XIC(ID86_MSG_ProcessAlarm.DN)[NOP() ,EQU(ID86_MSG_ProcessAlarm.Instance,1) [NEQ(MCP_00.MISC.ProcessAlarmData[0],MCP_00.IN.M01_UR20_16DI_P.ProcessAlarm.PRIT_OL) ,NEQ(MCP_00.MISC.ProcessAlarmData[1],MCP_00.IN.M01_UR20_16DI_P.ProcessAlarm.PRIT_UL) ,NEQ(MCP_00.MISC.ProcessAlarmData[2],MCP_00.IN.M01_UR20_16DI_P.ProcessAlarm.PRIT_US0) ,NEQ(MCP_00.MISC.ProcessAlarmData[3],MCP_00.IN.M01_UR20_16DI_P.ProcessAlarm.PRIT_US1) ] OTL(MCP_00.IN.M01_UR20_16DI_P.StatusProcessAlarm) CPS(MCP_00.MISC.ProcessAlarmData[0],MCP_00.IN.M01_UR20_16DI_P.ProcessAlarm,1) ,EQU(ID86_MSG_ProcessAlarm.Instance,2) [NEQ(MCP_00.MISC.ProcessAlarmData[0],MCP_00.IN.M02_UR20_16DI_P.ProcessAlarm.PRIT_OL) ,NEQ(MCP_00.MISC.ProcessAlarmData[1],MCP_00.IN.M02_UR20_16DI_P.ProcessAlarm.PRIT_UL) ,NEQ(MCP_00.MISC.ProcessAlarmData[2],MCP_00.IN.M02_UR20_16DI_P.ProcessAlarm.PRIT_US0) ,NEQ(MCP_00.MISC.ProcessAlarmData[3],MCP_00.IN.M02_UR20_16DI_P.ProcessAlarm.PRIT_US1) ] OTL(MCP_00.IN.M02_UR20_16DI_P.StatusProcessAlarm) CPS(MCP_00.MISC.ProcessAlarmData[0],MCP_00.IN.M02_UR20_16DI_P.ProcessAlarm,1) ,EQU(ID86_MSG_ProcessAlarm.Instance,3) [NEQ(MCP_00.MISC.ProcessAlarmData[0],MCP_00.IN.M03_UR20_4AI_UI_16.ProcessAlarm.PRIT_OL) ,NEQ(MCP_00.MISC.ProcessAlarmData[1],MCP_00.IN.M03_UR20_4AI_UI_16.ProcessAlarm.PRIT_UL) ,NEQ(MCP_00.MISC.ProcessAlarmData[2],MCP_00.IN.M03_UR20_4AI_UI_16.ProcessAlarm.PRIT_US0) ,NEQ(MCP_00.MISC.ProcessAlarmData[3],MCP_00.IN.M03_UR20_4AI_UI_16.ProcessAlarm.PRIT_US1) ] OTL(MCP_00.IN.M03_UR20_4AI_UI_16.StatusProcessAlarm) CPS(MCP_00.MISC.ProcessAlarmData[0],MCP_00.IN.M03_UR20_4AI_UI_16.ProcessAlarm,1) ,EQU(ID86_MSG_ProcessAlarm.Instance,4) [NEQ(MCP_00.MISC.ProcessAlarmData[0],MCP_00.IN.M04_UR20_16DO_P.ProcessAlarm.PRIT_OL) ,NEQ(MCP_00.MISC.ProcessAlarmData[1],MCP_00.IN.M04_UR20_16DO_P.ProcessAlarm.PRIT_UL) ,NEQ(MCP_00.MISC.ProcessAlarmData[2],MCP_00.IN.M04_UR20_16DO_P.ProcessAlarm.PRIT_US0) ,NEQ(MCP_00.MISC.ProcessAlarmData[3],MCP_00.IN.M04_UR20_16DO_P.ProcessAlarm.PRIT_US1) ] OTL(MCP_00.IN.M04_UR20_16DO_P.StatusProcessAlarm) CPS(MCP_00.MISC.ProcessAlarmData[0],MCP_00.IN.M04_UR20_16DO_P.ProcessAlarm,1) ,EQU(ID86_MSG_ProcessAlarm.Instance,5) [NEQ(MCP_00.MISC.ProcessAlarmData[0],MCP_00.IN.M05_UR20_16DO_P.ProcessAlarm.PRIT_OL) ,NEQ(MCP_00.MISC.ProcessAlarmData[1],MCP_00.IN.M05_UR20_16DO_P.ProcessAlarm.PRIT_UL) ,NEQ(MCP_00.MISC.ProcessAlarmData[2],MCP_00.IN.M05_UR20_16DO_P.ProcessAlarm.PRIT_US0) ,NEQ(MCP_00.MISC.ProcessAlarmData[3],MCP_00.IN.M05_UR20_16DO_P.ProcessAlarm.PRIT_US1) ] OTL(MCP_00.IN.M05_UR20_16DO_P.StatusProcessAlarm) CPS(MCP_00.MISC.ProcessAlarmData[0],MCP_00.IN.M05_UR20_16DO_P.ProcessAlarm,1) ,NOP() ];
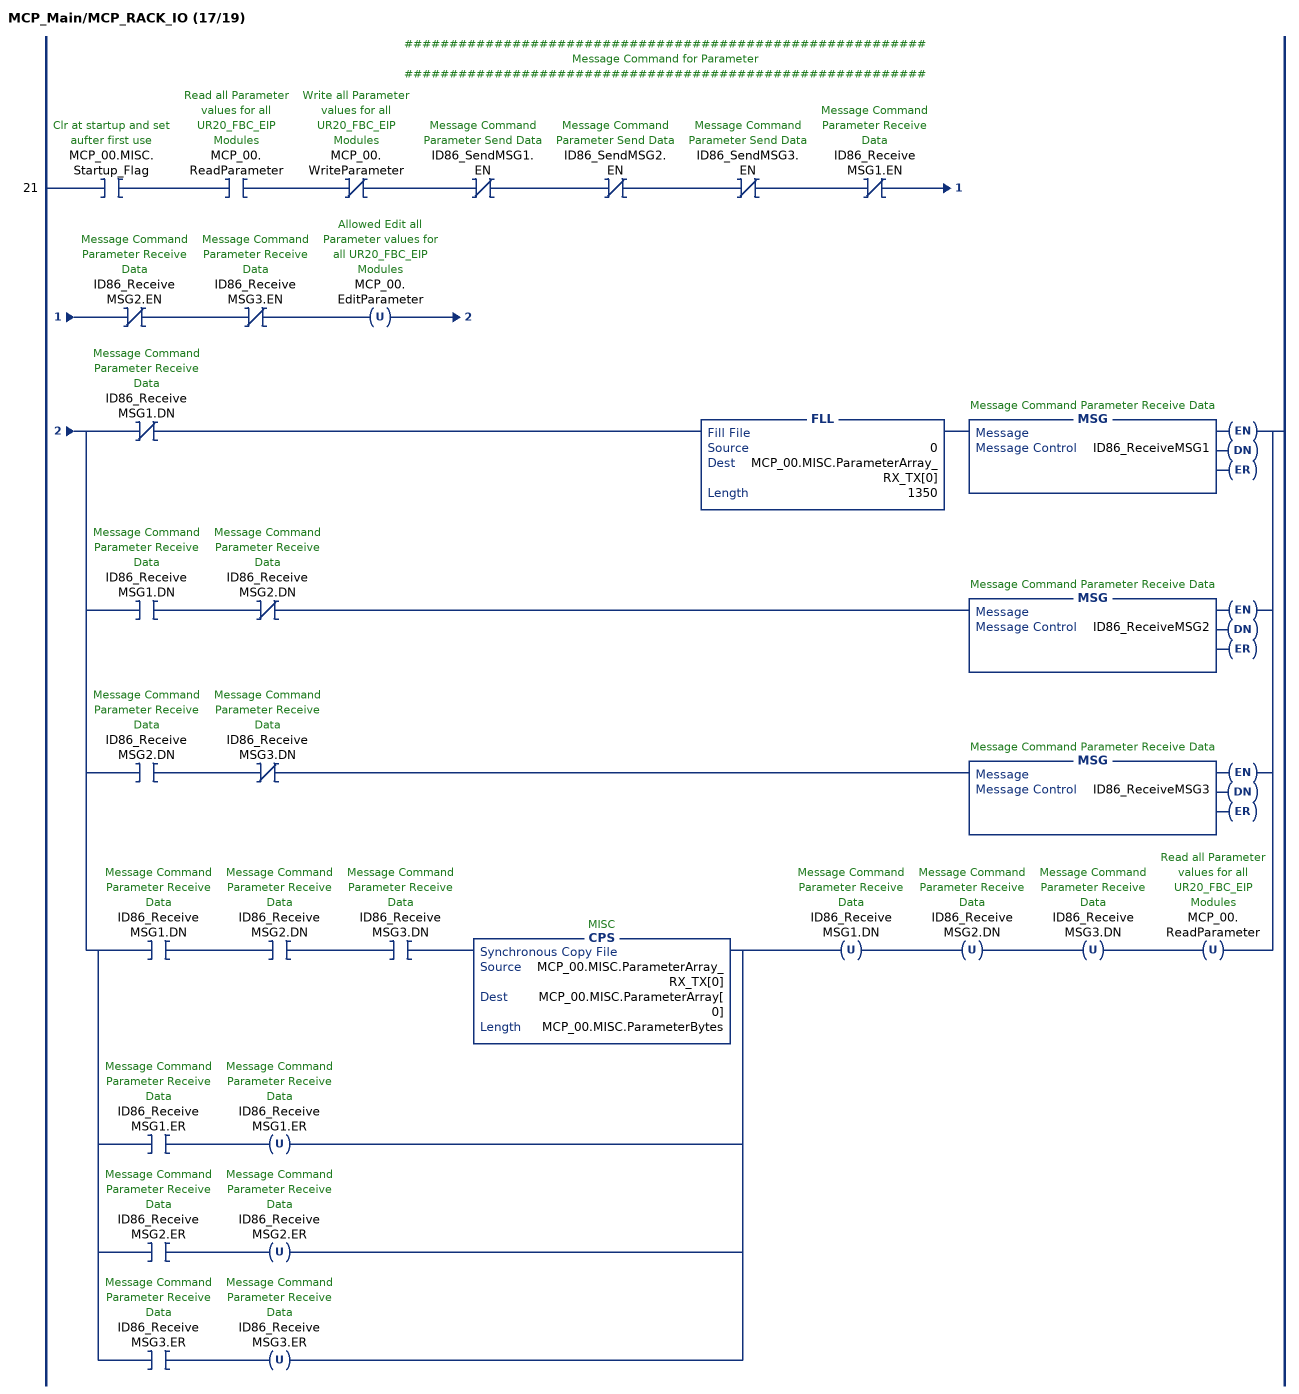
   // ##########################################################
   // Message Command for Parameter
   // ##########################################################
   21: XIC(MCP_00.MISC.Startup_Flag)XIC(MCP_00.ReadParameter)XIO(MCP_00.WriteParameter)XIO(ID86_SendMSG1.EN)XIO(ID86_SendMSG2.EN)XIO(ID86_SendMSG3.EN)XIO(ID86_ReceiveMSG1.EN)XIO(ID86_ReceiveMSG2.EN)XIO(ID86_ReceiveMSG3.EN)OTU(MCP_00.EditParameter)[XIO(ID86_ReceiveMSG1.DN) FLL(0,MCP_00.MISC.ParameterArray_RX_TX[0],1350) MSG(ID86_ReceiveMSG1) ,XIC(ID86_ReceiveMSG1.DN) XIO(ID86_ReceiveMSG2.DN) MSG(ID86_ReceiveMSG2) ,XIC(ID86_ReceiveMSG2.DN) XIO(ID86_ReceiveMSG3.DN) MSG(ID86_ReceiveMSG3) ,[XIC(ID86_ReceiveMSG1.DN) XIC(ID86_ReceiveMSG2.DN) XIC(ID86_ReceiveMSG3.DN) CPS(MCP_00.MISC.ParameterArray_RX_TX[0],MCP_00.MISC.ParameterArray[0],MCP_00.MISC.ParameterBytes) ,XIC(ID86_ReceiveMSG1.ER) OTU(ID86_ReceiveMSG1.ER) ,XIC(ID86_ReceiveMSG2.ER) OTU(ID86_ReceiveMSG2.ER) ,XIC(ID86_ReceiveMSG3.ER) OTU(ID86_ReceiveMSG3.ER) ] OTU(ID86_ReceiveMSG1.DN) OTU(ID86_ReceiveMSG2.DN) OTU(ID86_ReceiveMSG3.DN) OTU(MCP_00.ReadParameter) ];
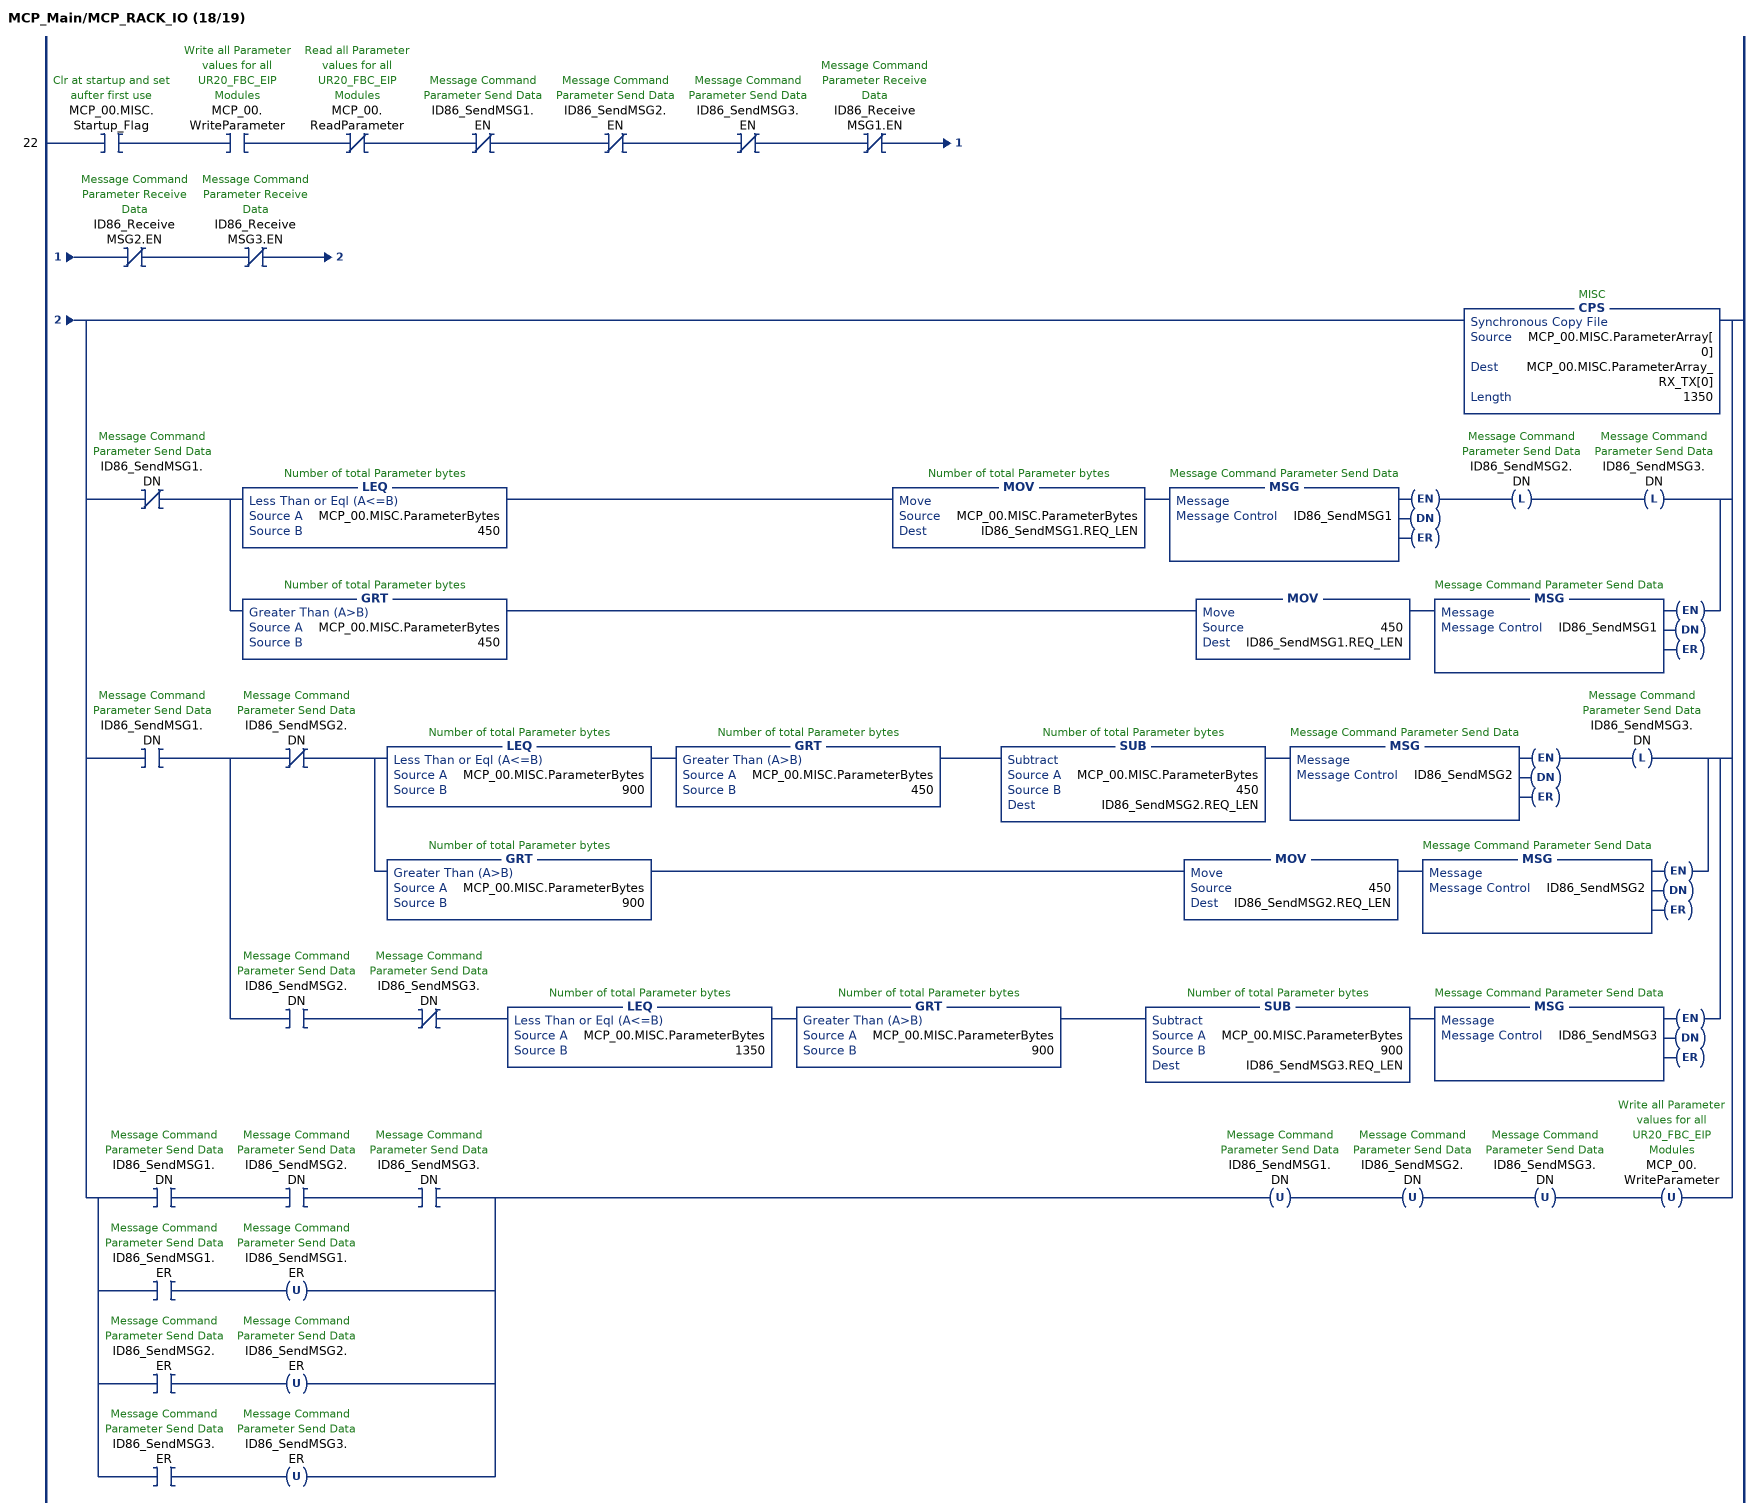
   22: XIC(MCP_00.MISC.Startup_Flag)XIC(MCP_00.WriteParameter)XIO(MCP_00.ReadParameter)XIO(ID86_SendMSG1.EN)XIO(ID86_SendMSG2.EN)XIO(ID86_SendMSG3.EN)XIO(ID86_ReceiveMSG1.EN)XIO(ID86_ReceiveMSG2.EN)XIO(ID86_ReceiveMSG3.EN)[CPS(MCP_00.MISC.ParameterArray[0],MCP_00.MISC.ParameterArray_RX_TX[0],1350) ,[XIO(ID86_SendMSG1.DN) [LEQ(MCP_00.MISC.ParameterBytes,450) MOV(MCP_00.MISC.ParameterBytes,ID86_SendMSG1.REQ_LEN) MSG(ID86_SendMSG1) OTL(ID86_SendMSG2.DN) OTL(ID86_SendMSG3.DN) ,GRT(MCP_00.MISC.ParameterBytes,450) MOV(450,ID86_SendMSG1.REQ_LEN) MSG(ID86_SendMSG1) ] ,XIC(ID86_SendMSG1.DN) [XIO(ID86_SendMSG2.DN) [LEQ(MCP_00.MISC.ParameterBytes,900) GRT(MCP_00.MISC.ParameterBytes,450) SUB(MCP_00.MISC.ParameterBytes,450,ID86_SendMSG2.REQ_LEN) MSG(ID86_SendMSG2) OTL(ID86_SendMSG3.DN) ,GRT(MCP_00.MISC.ParameterBytes,900) MOV(450,ID86_SendMSG2.REQ_LEN) MSG(ID86_SendMSG2) ] ,XIC(ID86_SendMSG2.DN) XIO(ID86_SendMSG3.DN) LEQ(MCP_00.MISC.ParameterBytes,1350) GRT(MCP_00.MISC.ParameterBytes,900) SUB(MCP_00.MISC.ParameterBytes,900,ID86_SendMSG3.REQ_LEN) MSG(ID86_SendMSG3) ] ,[XIC(ID86_SendMSG1.DN) XIC(ID86_SendMSG2.DN) XIC(ID86_SendMSG3.DN) ,XIC(ID86_SendMSG1.ER) OTU(ID86_SendMSG1.ER) ,XIC(ID86_SendMSG2.ER) OTU(ID86_SendMSG2.ER) ,XIC(ID86_SendMSG3.ER) OTU(ID86_SendMSG3.ER) ] OTU(ID86_SendMSG1.DN) OTU(ID86_SendMSG2.DN) OTU(ID86_SendMSG3.DN) OTU(MCP_00.WriteParameter) ] ];
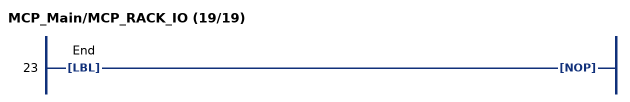
   23: LBL(End)NOP();
END_ROUTINE
